// TIA Portal project "read_old_project" (V15.1)

(* hardware
DEVICE "S7-1200 station_1"  S7-1200 Station
   slot 0: "Rack_0"  S7-1200 Rack  Rack  V1.0
   slot 1: "PLC_1"  CPU 1212C DC/DC/DC  6ES7 212-1AE40-0XB0  V4.2
      slot 3: "CB 1241 (RS485)"  CB 1241 (RS485)  6ES7 241-1CH30-1XB0  V1.0
*)

// ===== PLC "PLC_1"  CPU 1212C DC/DC/DC =====

VAR_GLOBAL   // PLC tag table "Default tag table"
   "I0" AT %I0.0 : Bool;
   "I1" AT %I0.1 : Bool;
   "I2" AT %I0.2 : Bool;
   "I3" AT %I0.3 : Bool;
   "distance_raw_1" AT %IW68 : Int;
   "distance_raw_2" AT %IW71 : Int;
   "Conv_power" AT %Q0.0 : Bool;
   "Conv_run" AT %Q0.1 : Bool;
   "Trigger_1" AT %M0.0 : Bool;
   "ChangeApp_1" AT %M0.1 : Bool;
   "AppNo_1" AT %MW2 : UInt;
   "Busy_1" AT %M1.0 : Bool;
   "Done_1" AT %M1.1 : Bool;
   "Error_1" AT %M1.2 : Bool;
   "Status_1" AT %MW4 : Word;
   "ExtStatus_1" AT %MW6 : Word;
   "ActAppNo_1" AT %MW8 : UInt;
   "RcvdLen_1" AT %MW10 : UInt;
   "Connect_1" AT %M0.7 : Bool;
   "Trigger_2" AT %M20.0 : Bool;
   "ChangeApp_2" AT %M20.1 : Bool;
   "Connect_2" AT %M20.7 : Bool;
   "Busy_2" AT %M21.0 : Bool;
   "Done_2" AT %M21.1 : Bool;
   "Error_2" AT %M21.2 : Bool;
   "AppNo_2" AT %MW22 : UInt;
   "Status_2" AT %MW24 : Word;
   "ExtStatus_2" AT %MW26 : Word;
   "ActAppNo_2" AT %MW28 : UInt;
   "RcvdLen_2" AT %MW30 : UInt;
   "System_Byte" AT %MB40 : Byte;
   "FirstScan" AT %M40.0 : Bool;
   "DiagStatusUpdate" AT %M40.1 : Bool;
   "AlwaysTRUE" AT %M40.2 : Bool;
   "AlwaysFALSE" AT %M40.3 : Bool;
   "Clock_Byte" AT %MB41 : Byte;
   "Clock_10Hz" AT %M41.0 : Bool;
   "Clock_5Hz" AT %M41.1 : Bool;
   "Clock_2.5Hz" AT %M41.2 : Bool;
   "Clock_2Hz" AT %M41.3 : Bool;
   "Clock_1.25Hz" AT %M41.4 : Bool;
   "Clock_1Hz" AT %M41.5 : Bool;
   "Clock_0.625Hz" AT %M41.6 : Bool;
   "Clock_0.5Hz" AT %M41.7 : Bool;
   "Edge_1" AT %M1000.0 : Bool;
   "Trigg" AT %M1000.1 : Bool;
   "clear" AT %M1000.2 : Bool;
   "distance_physic_1" AT %MW50 : Int;
   "distance_physic_2" AT %MW52 : Int;
   "M3.3" AT %M3.3 : Bool;
   "Tag_1" AT %M3.4 : Bool;
END_VAR

TYPE "Modbus_Register"
VERSION : 0.1
   STRUCT
      Camera_done : Int;
      Sensor_done : Int;
      Angle : DInt;
      Symetric : Int;
      Conveyor : Int;
      Reset : Int;
      Model : Int;
   END_STRUCT;
END_TYPE

DATA_BLOCK "O2D_Sensor_1"   // DB1
{ S7_Optimized_Access := 'TRUE' }
AUTHOR : ifm-sytl
FAMILY : O2Dxxx
NAME : O2Dxxx_TCP
VERSION : 3.1
// stored: InstanceOfName O2Dxxx_TCP
"O2Dxxx_TCP"
BEGIN
END_DATA_BLOCK

DATA_BLOCK "O2D_Sensor_2"   // DB2
{ S7_Optimized_Access := 'TRUE' }
AUTHOR : ifm-sytl
FAMILY : O2Dxxx
NAME : O2Dxxx_TCP
VERSION : 3.1
// stored: InstanceOfName O2Dxxx_TCP
"O2Dxxx_TCP"
BEGIN
END_DATA_BLOCK

DATA_BLOCK "O2D_Data"   // DB3
{ S7_Optimized_Access := 'TRUE' }
VERSION : 0.1
   VAR
      Response_Sensor_1 : Array[0..127] of Char;
      Response_Sensor_2 : Array[0..63] of Byte;
   END_VAR
BEGIN
END_DATA_BLOCK

DATA_BLOCK "DB_camera"   // DB4
{ S7_Optimized_Access := 'TRUE' }
VERSION : 0.1
   VAR
      Char_reponse : Array[0..127] of Char;
      data_save : Array[0..9] of DInt;
      model_save : Array[0..9] of Int;
      data_convert : DInt;
      data_convert_symetric : DInt;
      count : DInt;
      symetric : Int;
   END_VAR
BEGIN
END_DATA_BLOCK

DATA_BLOCK "DB_modbus"   // DB7
{ S7_Optimized_Access := 'FALSE' }
VERSION : 0.1
   VAR
      Register : "Modbus_Register";
      load_done : Bool;
      load_error : Bool;
      load_status : Word;
      slave_ndr : Bool;
      slave_dr : Bool;
      slave_error : Bool;
      slave_status : Word;
   END_VAR
BEGIN
   Register.Symetric := 1;
END_DATA_BLOCK

FUNCTION_BLOCK "O2Dxxx_TCP"   // FB1, SCL
{ S7_Optimized_Access := 'TRUE' }
AUTHOR : ifm-sytl
FAMILY : O2Dxxx
NAME : O2Dxxx_TCP
VERSION : 3.1
   VAR_INPUT
      LocIF_ID : UInt := 64;
      LocPortNo : UInt := 2000;
      RemIPAddr1 : USInt := 192;
      RemIPAddr2 : USInt := 168;
      RemIPAddr3 : USInt := 0;
      RemIPAddr4 : USInt := 49;
      RemPortNo : UInt := 50010;
      Connect : Bool;
      ConnID : UInt;
      TimeoutTime : Time := T#6S;
      Trigger : Bool;
      ChangeApp : Bool;
      AppNo : UInt := 1;
   END_VAR
   VAR_OUTPUT
      Busy : Bool := TRUE;
      Done : Bool;
      Error : Bool;
      Status : Word;
      ExtStatus : Word;
      ActAppNo : UInt;
      RcvdLen : UInt;
   END_VAR
   VAR_IN_OUT
      Data : Variant;
   END_VAR
   VAR
      fbSend : TSEND;
      fbReceive : TRCV_C;
      tonTimeoutCmd : TON_TIME;
      tonTimeoutPing : TON_TIME;
      tonDlyPing : TON_TIME;
      stConnSet : TCON_IP_v4;
      archRcvBuf : Array[0..33] of Char;
      archSendBuf : Array[0..39] of Char;
      iTicketID : Int;
      iTriggerRespLength : UInt;
      iActAppNo : UInt;
      iRdLength : UInt := 28;
      iRcvFunction : UInt;
      iLeftRcvLength : UInt;
      iBufSize : UInt;
      wStatus : Word;
      wErrorCode : Word;
      wExtErrorCode : Word;
      wErrorCodeConnect : Word;
      wErrorCodeSensor : Word;
      chUserCmdId : Char := '0';
      chCmdId : Char := '0';
      chRcvId : Char;
      xConnEstablished : Bool;
      xReqDisconnect : Bool;
      xReqReconnect : Bool;
      xSendPing : Bool;
      xInitExtRcvBuf : Bool;
      xUserAction : Bool;
      xSensorBlocked : Bool;
      xprevConnect : Bool;
      xprevTrigger : Bool;
      xprevChangeApp : Bool;
      xWaitResponse : Bool;
      xWaitPingResponse : Bool;
      xNewString : Bool;
      xWrToExtBuf : Bool;
      xRcvSysMssgToExt : Bool;
      xBusy : Bool;
      xError : Bool;
      xErrConnect : Bool;
      xErrTimeoutPing : Bool;
      xOutBusy : Bool := TRUE;
      xOutDone : Bool;
      xOutError : Bool;
   END_VAR
   VAR_TEMP
      DISizeOfExtRcvBuf : UDInt;
      DITemp : DInt;
      IDigitFactor : UInt;
      ITemp : Int;
      ICnt : UInt;
      WTemp : Word;
      CHInitValue : Char;
      BInitValue : Byte;
      BCmdId : Byte;
      ARBTemp : Array[0..2] of Byte;
      XRcvBufIsByte : Bool;
      XErrRcvBuf : Bool;
      XNdr : Bool;
      XSysMssgRcvd : Bool;
      XRcvdTicketMatch : Bool;
      XInitDataExch : Bool;
      XreTrigger : Bool;
      XreChangeApp : Bool;
      XErrASCII : Bool;
      XKeepOutput : Bool;
   END_VAR
BEGIN
   // Basic Application program for O2Dx
   // connected to S7 station via CPU-internal Ethernet interface
   // for S7-12xx CPU Firmware V4.1 or higher
   // for S7-15xx CPU Firmware V1.7 or higher

   // Function Block Version 3.1.00

   // With this FB you can
   // - establish TCP/IP V4 connection to the sensor
   // - trigger the sensor and read the result
   // - select active sensor application

   // ---- Inputs ----
   // LocIF_ID      : interface-ID of CPU Ethernet interface (refer to device configuration)
   // LocPortNo     : port.No. in CPU to use for this connection to the sensor (recommended 2000 ff.)
   // RemIPAddr1..4 : IP address of the sensor
   // RemPortNo     : port-No. of sensor process interface
   // Connect       : establish TCP connection to the sensor
   // ConnID        : unique ID as system reference for the connection to the sensor
   // TimeOutTime   : max. waiting time for response from the sensor
   // Trigger       : on rising edge send trigger command to sensor
   // ChangeApp, AppNo : on rising edge of ChangeApp
   //                    activate in AppNo assigned application-No. (3 digits) in the sensor

   // ---- Outputs ----
   // Busy          : no command accepted
   // Done          : command successful completed
   // Error         : error occurred
   // Status        : status information
   // ExtStatus     : extended status information
   // ActAppNo      : active sensor application-No.
   // RcvdLen       : data length in receive buffer

   // ---- In/Outputs ---
   // Data          : pointer to area where to store the data from the sensor


   // ******************************************************************************************************
   // Disclaimer of Warranties

   // ifm disclaims to the fullest extent authorized by law any and all warranties,
   // whether express or implied, including, without limitation,
   // any implied warranties of title, non-infringement, quiet enjoyment,
   // integration, merchantability or fitness for a particular purpose.

   // Without limitation of the foregoing, ifm expressly does not warrant that:
   // (a)  the software will meet your requirements or expectations;
   // (b)  the software or the software content will be free of bugs, errors,
   //      viruses or other defects;
   // (c)  any results, output, or data provided through or generated by the software
   //      will be accurate, up-to-date, complete or reliable;
   // (d)  the software will be compatible with third party software;
   // (e)  any errors in the software will be corrected


   // DEMO SOFTWARE AND TEMPLATES

   // Demo software and templates are provided “as is” and “as available”,
   // without any warranty of any kind, either express or implied.
   // The User acknowledges and agrees to use the software at User’s own risk.
   // In no event shall ifm be held liable for any direct, indirect, incidental
   // or consequential damages arising out of the use of or inability to use the software.
   // User may use the software solely for demonstration purposes
   // and to assess the software functionalities and capabilities.


   // Software written specifically for Customer

   // 1. The software created and used is put together by ifm specially to the customer
   //    using modular software components made by ifm for numerous applications (Standard software modules)
   //    and adapted to the contractual service required (customer-specific application program).

   // 2. Upon complete payment of the purchase price for the customer-specific application program,
   //    ifm transfers the non-exclusive, locally and temporarily unrestricted usage right
   //    thereof to the customer, without the customer acquiring any rights of any kind
   //    to the standard software module on which the individual or customer-specific adaptation is based.
   //    Notwithstanding these provisions, ifm reserves the right to produce and offer
   //    customer specific software solutions of the same kind for other customers
   //    based on other terms of reference. In any case ifm retains a simple right of usage
   //    of the customer–specific solution for internal purposes.

   // 3. Upon acceptance of the program, User acknowledges and agrees to use the software
   //    at User’s own risk. User also acknowledges and agrees upon acceptance of the program
   //    that the software meets the requirements of the specifications agreed upon.
   //    ifm disclaims any and all warranties, in particular regarding fitness of the software
   //    for a particular purpose.
   // ******************************************************************************************************


   // reset error signal
   #xError := #xError AND #xUserAction;  // initialize error signal if no user action active

   // read user inputs
   #XreTrigger := #Trigger AND NOT #xprevTrigger;  // rising edge of input TRIGGER
   #xprevTrigger := #Trigger;  // store state for edge detection
   #XreChangeApp := #ChangeApp AND NOT #xprevChangeApp;  // rising edge of input CHANGE APPLICATION
   #xprevChangeApp := #ChangeApp;  // store state for edge detection
   #xUserAction := (#XreTrigger OR #XreChangeApp) OR #xUserAction;  // set user action started

   // check if user inputs valid
   IF NOT #xError THEN  // no error occurred yet
     IF (#XreTrigger OR #XreChangeApp) AND #xOutBusy THEN
       // command input activated while output BUSY still active
       #xError := TRUE;
       #wErrorCode := 16#8301;  // set error code
       #wExtErrorCode := 0;
     ELSIF (#XreTrigger OR #XreChangeApp) AND NOT #Connect THEN
       // command input activated while input CONNECT = FALSE
       #xError := TRUE;
       #wErrorCode := 16#8302;  // set error code
       #wExtErrorCode := 0;
     ELSIF #XreTrigger AND #XreChangeApp THEN
       // command inputs activated simultaneously
       #xError := TRUE;
       #wErrorCode := 16#8303;  // set error code
       #wExtErrorCode := 0;
     END_IF;
   END_IF;  // check if user inputs valid

   // check external receive buffer is ARRAY OF CHAR or ARRAY OF BYTE
   #DISizeOfExtRcvBuf := CountOfElements(#Data);  // get size of external receive buffer
   #XErrRcvBuf := #DISizeOfExtRcvBuf = 0;  // check if external receive buffer is an array
   IF NOT #XErrRcvBuf THEN
     // external is an array
     #XRcvBufIsByte := TypeOfElements(#Data) = Byte;  // check if element data type of external receive buffer is BYTE
     #XErrRcvBuf := TypeOfElements(#Data) <> Char AND NOT #XRcvBufIsByte;  // check element data type of receive buffer is valid
   END_IF;
   IF #XErrRcvBuf AND NOT #xError THEN
     // external receive buffer invalid (only ARRAY of BYTE or ARRAY of CHAR are valid)
     #xError := TRUE;
     #wErrorCode := 16#8101;  // set error code
     #wExtErrorCode := 0;
   END_IF;

   // initialize external receive buffer
   #xInitExtRcvBuf := #XreTrigger OR #XreChangeApp OR #xInitExtRcvBuf;  // initialize external receive buffer
   IF #xInitExtRcvBuf AND NOT #XErrRcvBuf THEN
     #CHInitValue := ' ';  // set initial value for external receive buffer
     #BInitValue := 0;
     FOR #DITemp := 0 TO UDINT_TO_DINT(#DISizeOfExtRcvBuf) - 1 DO  // loop complete external receive buffer
       IF #XRcvBufIsByte THEN  // initialize external receive buffer with initial BYTE value
         #ITemp := MOVE_BLK_VARIANT(SRC := #BInitValue, SRC_INDEX := 0, DEST => #Data, DEST_INDEX := #DITemp, COUNT := 1);
       ELSE  // initialize external receive buffer with initial CHAR value
         #ITemp := MOVE_BLK_VARIANT(SRC := #CHInitValue, SRC_INDEX := 0, DEST => #Data, DEST_INDEX := #DITemp, COUNT := 1);
       END_IF;
       IF #ITemp <> 0 THEN  // error by access to external receive buffer
         IF NOT #xError THEN
           #xError := TRUE;
           #wErrorCode := 16#8400;  // set error code
           #wExtErrorCode := INT_TO_WORD(#ITemp);
         END_IF;
         EXIT;  // abort initialisation
       END_IF;
     END_FOR;
     #xInitExtRcvBuf := FALSE;  // reset request
   END_IF;  // initialize external receive buffer

   // set connection parameter
   IF #Connect AND NOT #xprevConnect THEN  // rising edge of input CONNECT
     // fill TCP/IP V4 connection structure
     #stConnSet.InterfaceId := #LocIF_ID;  // set hardware identifier of local interface (see CPU device properties )
     #stConnSet.ID := UINT_TO_WORD(#ConnID);  // set reference to this connection
     #stConnSet.ConnectionType := 17;  // set connection type = TCP
     #stConnSet.ActiveEstablished := TRUE;  // set active connection establishment
     #stConnSet.RemoteAddress.ADDR[1] := USINT_TO_BYTE(#RemIPAddr1);  // set IP address of remote connection partner
     #stConnSet.RemoteAddress.ADDR[2] := USINT_TO_BYTE(#RemIPAddr2);
     #stConnSet.RemoteAddress.ADDR[3] := USINT_TO_BYTE(#RemIPAddr3);
     #stConnSet.RemoteAddress.ADDR[4] := USINT_TO_BYTE(#RemIPAddr4);
     #stConnSet.RemotePort := #RemPortNo;  // set port address of remote connection partner
     #stConnSet.LocalPort := #LocPortNo;  // set local port address
   END_IF;  // rising edge of input CONNECT
   #xprevConnect := #Connect;  // store state for edge detection

   #xReqDisconnect := NOT #Connect AND #xConnEstablished OR #xReqDisconnect;  // set request to disconnect
   #xConnEstablished := #xConnEstablished AND NOT #xReqDisconnect AND NOT #xReqReconnect;  // reset connection established

   #fbReceive.CONT := #Connect AND NOT #xReqDisconnect AND NOT #xReqReconnect;  // establish connection
   #fbReceive.EN_R := TRUE;  // enable receive data
   #fbReceive.ADHOC := FALSE;  // disable AdHoc-mode
   #fbReceive.LEN := #iRdLength;  // set length to receive

   // receive data
   IF #xWrToExtBuf THEN  // select receive buffer
     // write to external receive buffer
     #fbReceive(CONNECT := #stConnSet,
                DATA := #Data);
   ELSE  // select receive buffer
     // write to internal receive buffer
     #fbReceive(CONNECT := #stConnSet,
                DATA := #archRcvBuf);
   END_IF;  // select receive buffer

   // result disconnect
   IF #fbReceive.STATUS = 16#7000 OR #fbReceive.STATUS = 16#0003 OR // disconnecting done
     #fbReceive.STATUS = 16#80A3  // no connection established
   THEN
     // disconnected successfully
     #xReqDisconnect := FALSE;  // reset request to disconnect
     #xReqReconnect := FALSE;  // reset request to reconnect
   END_IF;  // result disconnect

   // result connect
   IF NOT #Connect THEN  // reset error connect
     // reset error establish connection and timeout
     #xErrConnect := FALSE;
     #xErrTimeoutPing := FALSE;
     #xSensorBlocked := FALSE;
   ELSIF #fbReceive.CONT AND NOT #xConnEstablished AND #fbReceive.ERROR AND #fbReceive.STATUS <> 16#80C4 THEN
     // set error establish connection      
     #xErrConnect := TRUE;
     #xReqDisconnect := TRUE;
     #wErrorCodeConnect := #fbReceive.STATUS;  // save error code
   ELSIF #fbReceive.CONT AND NOT #xConnEstablished AND
     (#fbReceive.STATUS = 16#7004 OR #fbReceive.STATUS = 16#7006 OR #fbReceive.STATUS = 16#0001) THEN
     // connection established successfully
     #xConnEstablished := TRUE;
     #xErrConnect := FALSE;
     #xErrTimeoutPing := FALSE;
     #chCmdId := '1';  // execute command "v03"
   END_IF;  // result establish connection
   IF #xErrConnect AND NOT #xErrTimeoutPing AND NOT #xError THEN
     // set error code for error by establishing connection
     #xError := TRUE;
     #wErrorCode := 16#8201;  // set error code
     #wExtErrorCode := #wErrorCodeConnect;  // show error code of FB
   END_IF;  // error code establish connection

   // result receive data
   #XNdr := NOT #fbReceive.BUSY AND #fbReceive.DONE;  // new data received
   IF #fbReceive.CONT AND NOT #fbReceive.BUSY AND #fbReceive.ERROR THEN
     // error receive data
     #xReqReconnect := TRUE;  // set request disconnect
     IF NOT #xError AND #xBusy THEN
       #xError := TRUE;  // set error occurred
       #wErrorCode := 16#8203;  // set error code
       #wExtErrorCode := #fbReceive.STATUS;  // show error code of receive block
     END_IF;  // set error code
   END_IF;  // error receive data

   // cancel waiting for response
   IF NOT #fbReceive.CONT THEN
     #xWaitResponse := FALSE;
     #xWaitPingResponse := FALSE;
   END_IF;

   // timeout
   #tonTimeoutCmd(IN := #xWaitResponse AND #fbReceive.BUSY AND #xConnEstablished,
                  PT := #TimeoutTime);
   IF #tonTimeoutCmd.Q THEN
     // no response from sensor within surveillance time
     // (also happen if response string is shorter than expected;
     // the receive block will not provide data as long the buffer is not full yet)
     #xReqReconnect := TRUE;  // set request reconnect
     IF NOT #xError THEN
       #xError := TRUE;  // set error occurred
       #wErrorCode := 16#8205;  // set error code
       #wExtErrorCode := 0;
     END_IF;  // set error code
   END_IF;  // error receive data

   #XInitDataExch := NOT #xConnEstablished;  // preset request initialize data exchange

   IF #XNdr AND NOT #XInitDataExch THEN  // new data received

     #iLeftRcvLength := #iLeftRcvLength - UDINT_TO_UINT(#fbReceive.RCVD_LEN);  // update remaining length to receive

     CASE #iRcvFunction OF  // receive function selector

       0:  //receive 28 byte until "<CR><LF>10" received
         // look for "<CR><LF>10" in received data;
         // if found activate receive byte-wise

         FOR #ITemp := 0 TO 24 DO  // 25 possible DWORDs to check
           IF #archRcvBuf[#ITemp] = '$R' AND #archRcvBuf[#ITemp + 1] = '$L' AND
             #archRcvBuf[#ITemp + 2] = '1' AND #archRcvBuf[#ITemp + 3] = '0' THEN  // "<CR><LF>10" found

             // prepare FOR receiving the rest Byte-wise
             #xWaitResponse := FALSE;
             #iRdLength := 1;  // set length to receive
             #iRcvFunction := 1;  // activate receive function 1
           END_IF;  // "<CR><LF>10" found
         END_FOR;  // 25 possible DWORDs to check

       1:  // receive byte-wise until protocol V03 approved
         // check for response = ..."1003*<CR><LF>" to confirm protocol V03 is active

         #archRcvBuf[28] := #archRcvBuf[0];  // copy received byte to end of received data

         // shift received data in buffer 1 byte to left
         FOR #ITemp := 0 TO 27 DO
           #archRcvBuf[#ITemp] := #archRcvBuf[#ITemp + 1];
         END_FOR;

         // check for "1003" and "<CR><LF>"
         IF #archRcvBuf[21] = '1' AND #archRcvBuf[22] = '0' AND #archRcvBuf[23] = '0' AND #archRcvBuf[24] = '3' AND
           #archRcvBuf[26] = '$R' AND #archRcvBuf[27] = '$L' THEN  // "1003" and "<CR><LF>" received

           // response to command "v03" received
           IF #archRcvBuf[25] <> '*' THEN  // check acknowledge
             // protocol V03 not acknowledged
             IF NOT #xError THEN  // error protocol V03
               #xError := TRUE;
               #wErrorCode := 16#8001;  // set error code
               #wExtErrorCode := 0;
             END_IF;  // error protocol V03
             #XInitDataExch := TRUE;
           ELSE  // check acknowledge
             // protocol V03 acknowledged
             #chCmdId := '8';  // execute command "a?"
             #iLeftRcvLength := 0;  // no more data to receive
             #iRcvFunction := 4;  // complete command
           END_IF;  // check acknowledge

         END_IF;  // "1003" and "<CR><LF>" received

       2:  // evaluate ID and length information
         // identify length information and response-ID;
         // check if payload is to receive with or without evaluation

         #XErrASCII := #archRcvBuf[4] <> 'L' OR
         #archRcvBuf[5] <> '0' OR #archRcvBuf[6] <> '0' OR #archRcvBuf[7] <> '0' OR #archRcvBuf[8] <> '0' OR
         #archRcvBuf[15] <> '$L';  // check begin and end of length information string

         // convert length from ASCII to UINT
         #IDigitFactor := 10000;  // set digit factor
         #iLeftRcvLength := 0;  // initialize remaining length to receive
         FOR #ITemp := 9 TO 13 DO  // loop lowest 5 length information digits
           IF #archRcvBuf[#ITemp] < '0' OR #archRcvBuf[#ITemp] > '9' THEN  // check for ASCII range 0..9
             // out of range
             #XErrASCII := TRUE;  // set error ASCII data
           ELSE  // check for ASCII range 0..9
             // calculate response length
             #iLeftRcvLength := (CHAR_TO_UINT(#archRcvBuf[#ITemp]) - 48) * #IDigitFactor + #iLeftRcvLength;
           END_IF;  // check for ASCII range 0..9
           #IDigitFactor := #IDigitFactor / 10;  // update digit factor for next digit
         END_FOR; // loop lowest 5 length information digits

         IF #XErrASCII THEN  // error in length information data
           // error in ASCII data of length information string
           IF NOT #xError THEN  // no error yet
             #xError := TRUE;
             #wErrorCode := 16#8402;  // set error code
             #wExtErrorCode := 0;
           END_IF;  // no error yet
           // synchronize data exchange
           #XInitDataExch := TRUE;  // enable initialize data exchange
           #chCmdId := '1';  // execute command "v03"
         ELSE  // error in length information data
           // length information extracted successfully
           // prepare to receive payload data

           // correct left length to receive
           #iLeftRcvLength := #iLeftRcvLength - 4;  // 4 Byte ticket-No. is received already

           // evaluate received command-ID and ticket-No.
           #chRcvId := #archRcvBuf[0];  // store received command-ID
           #XSysMssgRcvd := #archRcvBuf[0] = '0' AND #archRcvBuf[1] = '0' AND #archRcvBuf[2] = '0' AND #archRcvBuf[3] = '0';  // check response-ID
           #XRcvdTicketMatch := #archRcvBuf[0] = #archSendBuf[0] AND
           #archRcvBuf[1] = #archSendBuf[1] AND
           #archRcvBuf[2] = #archSendBuf[2] AND
           #archRcvBuf[3] = #archSendBuf[3];  // received ticket-No. match to last sent ticket-No.
           #xWaitResponse := #xWaitResponse AND NOT #XRcvdTicketMatch;  // reset wait for response if response of command is received

           // select receive buffer for payload data to receive
           #xRcvSysMssgToExt := #XSysMssgRcvd AND NOT #xSensorBlocked AND NOT #Trigger AND NOT #ChangeApp AND NOT #xError;
           #xInitExtRcvBuf := (#xRcvSysMssgToExt OR #XRcvdTicketMatch AND #chRcvId = '9') AND NOT #XErrRcvBuf;
           #xWrToExtBuf := #xInitExtRcvBuf AND #iLeftRcvLength <> 3;
           IF #xWrToExtBuf THEN  // select receive buffer
             // use external receive buffer
             #iBufSize := UDINT_TO_UINT(#DISizeOfExtRcvBuf);  // set receive buffer size to size of external buffer
             #iTriggerRespLength := #iLeftRcvLength;  // store received payload data length
           ELSE  // select receive buffer
             // use internal receive buffer
             #iBufSize := 34;  // set receive buffer size to size of internal buffer
             #iTriggerRespLength := 0;  // initialize received payload data length
           END_IF;  // select receive buffer

           #iRdLength := MIN(IN1 := #iLeftRcvLength, IN2 := #iBufSize);  // limit receive length to receive buffer size
           #xNewString := TRUE;  // set new string will be received

           // select next receive function
           IF NOT #XRcvdTicketMatch AND NOT #xSensorBlocked OR #xWrToExtBuf THEN
             #iRcvFunction := 4;  // receive data without evaluation
           ELSE
             #iRcvFunction := 3;  // receive data to evaluate
           END_IF;  // select next receive function

         END_IF;  // error in length information data

       3:  // evaluate response data
         IF #chRcvId = '0' THEN
           // ping response received
           IF NOT #xUserAction AND #archRcvBuf[0] = '!' THEN
             // sensor used by another application (GUI)
             #xSensorBlocked := TRUE;
           ELSIF NOT #xUserAction THEN
             // sensor available
             IF #xSensorBlocked THEN  // sensor was unavailable
               #chCmdId := '8';  // execute command "a?"
               #xSensorBlocked := FALSE;
             END_IF;  // sensor available
           END_IF;  // ping response received

         ELSIF #fbReceive.RCVD_LEN = 3 AND #archRcvBuf[0] = '?' AND #archRcvBuf[1] = '$R' AND #archRcvBuf[2] = '$L' THEN
           // sensor returns "command unknown"
           IF NOT #xError THEN
             // error command unknown
             #xError := TRUE;
             #wErrorCode := 16#8300;  // set error code
             #wExtErrorCode := 0;
           END_IF;  // error command unknown

         ELSIF #fbReceive.RCVD_LEN = 3 AND #archRcvBuf[0] = '!' AND #archRcvBuf[1] = '$R' AND #archRcvBuf[2] = '$L' THEN
           // sensor returns "unable to execute command"
           // get error code from sensor
           #chCmdId := '2';  // execute command "E?"
         ELSE
           // data to evaluate received
           // evaluate received data of each command special
           CASE CHAR_TO_INT(#chRcvId) - 48 OF  // convert ASCII to integer

             2:  // evaluate response to command "E?"
               // error code from sensor received
               #wErrorCodeSensor.%B1 := INT_TO_BYTE((CHAR_TO_INT(#archRcvBuf[0]) - 48) * 16 + (CHAR_TO_INT(#archRcvBuf[1]) - 48));  // convert hi-byte of error code
               #wErrorCodeSensor.%B0 := INT_TO_BYTE((CHAR_TO_INT(#archRcvBuf[2]) - 48) * 16 + (CHAR_TO_INT(#archRcvBuf[3]) - 48));  // convert low-byte of error code
               IF #xUserAction AND NOT #xError THEN
                 // error sensor unable to execute command
                 #xError := TRUE;
                 #wErrorCode := 16#8000;  // set error code
                 #wExtErrorCode := #wErrorCodeSensor;  // show error code from sensor
               END_IF;  // error sensor unable to execute command
               #chCmdId := '8';  // execute command "a?"

             4:  // evaluate response to command "c + group and application-No."
               #chCmdId := '8';  // execute command "a?"

             8:  // evaluate response to command "a?"
               // extract number of active configuration and convert ASCII to integer
               #iActAppNo := (CHAR_TO_UINT(#archRcvBuf[5]) - 48) * 10 + CHAR_TO_UINT(#archRcvBuf[6]) - 48;

             9:  // evaluate response to command "T?"
               // response length = 3 characters but not a negative acknowledge;
               // then copy received data into external receive buffer
               IF #XRcvBufIsByte THEN  // element data type of external receive buffer is BYTE
                 // convert data type and copy to external receive buffer
                 #ARBTemp[0] := CHAR_TO_BYTE(#archRcvBuf[0]);
                 #ARBTemp[1] := CHAR_TO_BYTE(#archRcvBuf[1]);
                 #ARBTemp[2] := CHAR_TO_BYTE(#archRcvBuf[2]);
                 #ITemp := MOVE_BLK_VARIANT(SRC := #ARBTemp, SRC_INDEX := 0, DEST => #Data, DEST_INDEX := 0, COUNT := 3);
               ELSE  // copy to external receive buffer
                 #ITemp := MOVE_BLK_VARIANT(SRC := #archRcvBuf, SRC_INDEX := 0, DEST => #Data, DEST_INDEX := 0, COUNT := 3);
               END_IF;
               IF #ITemp = 0 THEN  // copy data successful
                 #iTriggerRespLength := 3;  // store received payload data length
               ELSIF NOT #xError THEN
                 // error by access to external receive buffer
                 #xError := TRUE;
                 #wErrorCode := 16#8400;  // set error code
                 #wExtErrorCode := INT_TO_WORD(#ITemp);
               END_IF;

           END_CASE;  // evaluate received data of each command special
         END_IF;  // evaluate response data
         #iRcvFunction := 4;  // evaluation finished, receive rest of response data

     END_CASE;  // receive function selector

     // receive data without evaluation
     IF #iRcvFunction = 4 AND NOT #XInitDataExch THEN  // receive function 4 active

       // receive data without evaluation
       IF #iLeftRcvLength > 0 THEN  // receiving data completed?
         // not all data received yet
         IF NOT #xNewString AND #xWrToExtBuf THEN
           // external buffer full
           IF NOT #xError THEN  // error external receive buffer too small
             #xError := TRUE;
             #wErrorCode := 16#8401;  // set error code
             #wExtErrorCode := UINT_TO_WORD(#iTriggerRespLength);  // show trigger response length
           END_IF;  // error external receive buffer too small
           #xWrToExtBuf := FALSE;  // change to internal receive buffer
           #iBufSize := 34;  // set size of used buffer
         END_IF;  // external buffer full
         #iRdLength := MIN(IN1 := #iLeftRcvLength, IN2 := #iBufSize);  // limit receive length
         #xNewString := FALSE;  // reset new string to receive

       ELSE  // receiving data completed?
         // all data received
         #xWrToExtBuf := FALSE;  // activate internal receive buffer
         #xBusy := #xBusy AND (#xWaitResponse OR #chRcvId = '0');  // enable new command, except Ping response is received
         #iRdLength := 20;  // set length 16 byte length information string + 4 byte ticket-No.
         #iRcvFunction := 2;  // activate receive function 2
       END_IF;  // receiving data completed?
     END_IF;  // receive function 4 active

   END_IF;  // new data received

   // initialize data exchange
   IF #XInitDataExch THEN
     // prepare for receiving response to command "v03"
     #xBusy := FALSE;
     #xWrToExtBuf := FALSE;
     #xRcvSysMssgToExt := FALSE;
     #iRdLength := 28; // set initial length to read
     #iRcvFunction := 0;  // activate receive function 0
   END_IF;  // initialize data exchange

   //**************************************************************
   // after certain time of inactivity send ping command to check connection
   #tonDlyPing(IN := (#iRcvFunction = 2 OR #xSensorBlocked) AND #fbReceive.BUSY AND NOT #xBusy AND NOT #xSendPing,
               PT := t#3s,  // inactivity time
               Q => #xSendPing);  // activate send ping command

   // timeout ping
   #xWaitPingResponse := #xWaitPingResponse AND NOT #XNdr AND #xConnEstablished;  // any received data reset ping timeout
   #tonTimeoutPing(IN := #xWaitPingResponse,
                   PT := t#1s);
   IF #tonTimeoutPing.Q THEN
     #xErrTimeoutPing := TRUE;  // timeout ping occurred
     #xReqReconnect := TRUE;  // set request reconnect
   END_IF;
   IF #xErrTimeoutPing AND NOT #xError THEN  // error timeout ping
     #xError := TRUE;  // set error occurred
     #wErrorCode := 16#8206;  // set error code
     #wExtErrorCode := 0;
   END_IF;  // error timeout ping

   //**************************************************************
   // request send command
   IF #XreTrigger THEN
     #chUserCmdId := '9';  // store user requested command-ID
   END_IF;
   IF #XreChangeApp THEN
     #chUserCmdId := '4';  // store user requested command-ID
   END_IF;
   IF (#XreTrigger OR #XreChangeApp) AND NOT #xError THEN
     #chCmdId := #chUserCmdId;  // apply requested command
   END_IF;
   #xBusy := #chCmdId <> '0' OR #xBusy;  // if command requested then set busy

   #fbSend.REQ := (#chCmdId <> '0' OR #xSendPing) AND #xConnEstablished AND NOT #fbSend.BUSY;  // activate sending data
   IF #fbSend.REQ THEN  // build command to send

     // create new ticket-ID
     IF #iTicketID > 0 AND #iTicketID < 999 THEN
       #iTicketID := #iTicketID + 1;  // increase ticket-ID
     ELSE  // limit reached
       #iTicketID := 1;  // initialize ticket-ID
     END_IF;

     // fill most common parts into send buffer
     #archSendBuf[0] := #chCmdId;  // command-ID
     #archSendBuf[1] := INT_TO_CHAR(#iTicketID / 100 + 48);  // convert 100th digit of ticket-ID to ASCII
     #ITemp := #iTicketID - #iTicketID / 100 * 100;  // get rest of division
     #archSendBuf[2] := INT_TO_CHAR(#ITemp / 10 + 48);  // convert 10th digit of ticket-ID to ASCII
     #ITemp := #ITemp - #ITemp / 10 * 10;  // get rest of division
     #archSendBuf[3] := INT_TO_CHAR(#ITemp + 48);  // convert 1th digit of ticket-ID to ASCII
     #archSendBuf[4] := 'L';
     FOR #ITemp := 5 TO 12 DO  // preset length information with "0"
       #archSendBuf[#ITemp] := '0';
     END_FOR;
     #archSendBuf[13] := '8';  // preset most common command length = 8 bytes
     #archSendBuf[14] := '$R';  // "<CR>"
     #archSendBuf[15] := '$L';  // "<LF>"
     #archSendBuf[16] := #archSendBuf[0];  // repeat ticket-No.
     #archSendBuf[17] := #archSendBuf[1];
     #archSendBuf[18] := #archSendBuf[2];
     #archSendBuf[19] := #archSendBuf[3];
     FOR #ITemp := 20 TO 39 DO  // preset rest of send buffer with " "
       #archSendBuf[#ITemp] := ' ';
     END_FOR;

     // select command
     CASE CHAR_TO_INT(#chCmdId) - 48 OF  // convert ASCII to integer

       0:  // command "s?" as ping command 
         #archSendBuf[20] := 's';
         #archSendBuf[21] := '?';
         #archSendBuf[22] := '$R';  // "<CR>"
         #archSendBuf[23] := '$L';  // "<LF>"
         #fbSend.LEN := 24;  // set length to send

       1:  // command "v03" in all protocol versions
         // "v03<CR><LF>" for protocol 1 and 4
         // "1002v03<CR><LF>" for protocol 2
         // "1003L000000009<CR><LF>1003v03<CR><LF>" for protocol 3
         Strg_TO_Chars(Strg := 'v03$R$L1002v03$R$L1003L000000009$R$L1003v03$R$L',  // source string
                       Chars := #archSendBuf,  // destination array
                       pChars := 0,  // destination start index
                       Cnt => #ICnt);  // number of copied characters
         #fbSend.LEN := UINT_TO_UDINT(#ICnt);  // set length to send

       2:  // command "E?"
         #archSendBuf[20] := 'E';
         #archSendBuf[21] := '?';
         #archSendBuf[22] := '$R';  // "<CR>"
         #archSendBuf[23] := '$L';  // "<LF>"
         #fbSend.LEN := 24;  // set length to send

       4:  // command "c + group-No. + application-No."
         #archSendBuf[12] := '1';  // overwrite preset payload data length
         #archSendBuf[13] := '0';  // command length = 10 bytes
         #archSendBuf[20] := 'c';
         #archSendBuf[21] := UINT_TO_CHAR(#AppNo / 100 + 48);  // convert 100th digit of input APPLICATION-NO. to ASCII
         #ITemp := UINT_TO_INT(#AppNo - #AppNo / 100 * 100);  // get rest of division
         #archSendBuf[22] := INT_TO_CHAR(#ITemp / 10 + 48);  // convert 10th digit of APPLICATION-NO. to ASCII
         #ITemp := #ITemp - #ITemp / 10 * 10;  // get rest of division
         #archSendBuf[23] := INT_TO_CHAR(#ITemp + 48);  // convert 1th digit of APPLICATION-NO. to ASCII
         #archSendBuf[24] := '$R';  // "<CR>"
         #archSendBuf[25] := '$L';  // "<LF>"
         #fbSend.LEN := 26;  // set length to send

       8:  // command "a?"
         #archSendBuf[20] := 'a';
         #archSendBuf[21] := '?';
         #archSendBuf[22] := '$R';  // "<CR>"
         #archSendBuf[23] := '$L';  // "<LF>"
         #fbSend.LEN := 24;  // set length to send

       9:  // command "T?"
         #archSendBuf[20] := 'T';
         #archSendBuf[21] := '?';
         #archSendBuf[22] := '$R';  // "<CR>"
         #archSendBuf[23] := '$L';  // "<LF>"
         #fbSend.LEN := 24;  // set length to send

       ELSE  // unknown command-ID
         #fbSend.REQ := FALSE;  // reset send request
     END_CASE;  // select command

     // command is build
     #xWaitPingResponse := #fbSend.REQ AND #chCmdId = '0';  // set wait for ping response
     #xWaitResponse := #fbSend.REQ AND NOT #xWaitPingResponse;  // set wait for command response
     #chCmdId := '0';  // initialize command-ID
   END_IF;  // build command to send

   // send data
   #fbSend(ID := #stConnSet.ID,
           DATA := #archSendBuf);  // send data

   // check send result
   IF #fbSend.ERROR AND #archSendBuf[0] <> '0' THEN
     // error while sending data
     #xReqReconnect := TRUE;  // set request reconnect
     IF NOT #xError THEN
       #xError := TRUE;
       #wErrorCode := 16#8204;  // set error code
       #wExtErrorCode := #fbSend.STATUS;  // show error code of send block
     END_IF;  // send error
   END_IF;  // send result

   // build internal status code
   IF NOT #Connect AND (#fbReceive.STATUS = 16#7000 OR #fbReceive.STATUS = 16#0003) THEN
     #wStatus := 16#1000;  // disconnected
   ELSIF #xReqDisconnect OR #xReqReconnect THEN
     #wStatus := 16#1001;  // disconnecting in progress
   ELSIF #Connect AND NOT #xConnEstablished THEN
     #wStatus := 16#1002;  // connecting in progress
   ELSIF #iRcvFunction < 2 THEN
     // synchronisation phase
     IF #fbSend.BUSY THEN
       #wStatus := 16#2001;  // send command "v03"
     ELSIF #iRcvFunction = 0 THEN
       #wStatus := 16#2002;
     ELSE
       #wStatus := 16#2003;
     END_IF;
     // end synchronisation phase
   ELSIF #xSensorBlocked THEN
     #wStatus := 16#3000;  // sensor unavailable
   ELSE
     // data exchange phase
     IF NOT #xBusy AND #iRcvFunction = 2 THEN
       #wStatus := 16#7000;
     ELSIF #fbSend.BUSY THEN
       #wStatus := 16#7001;  // send data active
     ELSE
       #wStatus := 16#7000 OR UINT_TO_WORD(#iRcvFunction);
     END_IF;
     IF #xBusy THEN
       #BCmdId := INT_TO_BYTE(CHAR_TO_INT(#archSendBuf[0]) - 48);  // convert ASCII to byte
       #wStatus.%B1 := #wStatus.%B1 OR #BCmdId;  // add active command-ID
     END_IF;
     // end data exchange phase
   END_IF;  // build internal status code

   // output BUSY
   #xOutBusy := #xBusy OR #iRcvFunction < 2 OR NOT #xConnEstablished OR #xReqReconnect OR #xSensorBlocked;
   #Busy := #xOutBusy;

   // keep output DONE and ERROR as long the triggering input still active
   #XKeepOutput := (#chUserCmdId = '9' AND #Trigger OR #chUserCmdId = '4' AND #ChangeApp) AND NOT #XreTrigger AND NOT #XreChangeApp;

   // output DONE
   #xOutDone := (#iRcvFunction = 2 AND #xRcvSysMssgToExt  // receive system message to ext. buffer finished
   OR #xUserAction  // user action started
   ) AND NOT #xBusy AND NOT #xError AND NOT #XErrRcvBuf // no command in progress and no error
   OR #xOutDone AND #XKeepOutput;  // keep output as long triggering input still set
   #Done := #xOutDone;

   // output ERROR
   #xOutError := (#xError OR #XErrRcvBuf) AND NOT #xBusy AND NOT #xOutDone  // error occurred and no command in progress
   OR #xOutError AND #XKeepOutput;  // keep output as long triggering input still set
   #Error := #xOutError;

   // output STATUS and EXTSTATUS
   IF #xOutDone THEN
     // if output DONE is set, show STATUS = 0x0000, EXTSTATUS = internal status code
     #Status := 16#0000;
     #ExtStatus := #wStatus;
   ELSIF #xOutError THEN
     // if output ERROR is set, show error codes STATUS and EXTSTATUS
     #Status := #wErrorCode;
     #ExtStatus := #wExtErrorCode;
   ELSE
     // else show STATUS = internal status code, EXTSTATUS = status of receive block
     #Status := #wStatus;
     #ExtStatus := #fbReceive.STATUS;
   END_IF;  // end output STATUS

   // output ACTIVE APPLICATION-NO. in the sensor
   IF NOT #xConnEstablished OR #xSensorBlocked THEN
     #iActAppNo := 0;  // reset active application 
   END_IF;
   #ActAppNo := #iActAppNo;

   // output DATA LENGTH in external receive buffer
   IF #XreTrigger OR #XreChangeApp OR #xInitExtRcvBuf OR #XErrRcvBuf THEN
     #RcvdLen := 0;
   ELSIF #xOutDone AND (#xUserAction OR #xRcvSysMssgToExt) THEN
     #RcvdLen := #iTriggerRespLength;
   END_IF;

   #xUserAction := #xUserAction AND #xBusy;  // reset user action started

   // reset receive system message to external receive buffer
   #xRcvSysMssgToExt := #xRcvSysMssgToExt AND NOT #xOutDone;  // reset if output DONE is set
END_FUNCTION_BLOCK

FUNCTION "Angle_Convert_Push" : Void   // FC1, LAD
{ S7_Optimized_Access := 'TRUE' }
VERSION : 0.1
   VAR_TEMP
      Temp_1 : DInt;
      Temp_2 : DInt;
      Temp_3 : DInt;
      Temp_4 : DInt;
      Temp_5 : DInt;
      Temp_6 : DInt;
   END_VAR
BEGIN

REGION Network 1 (SCL)
   //Convert
   #Temp_1 := CHAR_TO_DINT("DB_camera".Char_reponse[33]);
   #Temp_2 := CHAR_TO_DINT("DB_camera".Char_reponse[34]);
   #Temp_3 := CHAR_TO_DINT("DB_camera".Char_reponse[35]);
   #Temp_4 := CHAR_TO_DINT("DB_camera".Char_reponse[36]);
   #Temp_5 := CHAR_TO_DINT("DB_camera".Char_reponse[37]);
   #Temp_6 := CHAR_TO_DINT("DB_camera".Char_reponse[38]);

   "DB_camera".data_convert := (#Temp_2 - 48) * 10000000 + (#Temp_3 - 48) * 1000000 + (#Temp_4 - 48) * 100000 + (#Temp_6 - 48) * 10000;
   IF #Temp_1 = 43 THEN
       "DB_camera".data_convert := "DB_camera".data_convert * (-1);
   END_IF;
   //Push //symetric 1=rectang//2=square
   IF ("DB_camera".data_convert >= -18000000) AND ("DB_camera".data_convert <= 18000000) THEN
       #Temp_1 := CHAR_TO_DINT("DB_camera".Char_reponse[33]);
       IF "DB_modbus".Register.Symetric = 0 THEN
           "DB_camera".data_convert_symetric := "DB_camera".data_convert;
       ELSIF "DB_modbus".Register.Symetric = 1 THEN
           IF "DB_camera".data_convert > 9000000 THEN
               "DB_camera".data_convert_symetric := "DB_camera".data_convert - 18000000;
           ELSIF "DB_camera".data_convert < -9000000 THEN
               "DB_camera".data_convert_symetric := "DB_camera".data_convert + 18000000;
           ELSE
               "DB_camera".data_convert_symetric := "DB_camera".data_convert;
           END_IF;
       ELSIF "DB_modbus".Register.Symetric = 2 THEN
           IF "DB_camera".data_convert > 4500000 AND "DB_camera".data_convert <= 13500000 THEN
               "DB_camera".data_convert_symetric := "DB_camera".data_convert - 9000000;
           ELSIF "DB_camera".data_convert < -4500000 AND "DB_camera".data_convert >= -13500000 THEN
               "DB_camera".data_convert_symetric := "DB_camera".data_convert + 9000000;
           ELSIF "DB_camera".data_convert > 13500000 THEN
               "DB_camera".data_convert_symetric := "DB_camera".data_convert - 18000000;
           ELSIF "DB_camera".data_convert < -13500000 THEN
               "DB_camera".data_convert_symetric := "DB_camera".data_convert + 18000000;
           ELSE
               "DB_camera".data_convert_symetric := "DB_camera".data_convert;
           END_IF; 
       END_IF;

       "DB_camera".count := "DB_camera".count + 1;
       "DB_camera".data_save["DB_camera".count - 1] := "DB_camera".data_convert_symetric;
       "DB_camera".model_save["DB_camera".count - 1] := CHAR_TO_DINT("DB_camera".Char_reponse[21]) - 48;
   END_IF;
END_REGION
END_FUNCTION

FUNCTION "Angle_Mov_Pull" : Void   // FC2, LAD
{ S7_Optimized_Access := 'TRUE' }
VERSION : 0.1
   VAR_TEMP
      forloop : DInt;
   END_VAR
BEGIN

REGION Network 1 (SCL)
   IF ("DB_camera".data_save[0] >= -18000000) AND ("DB_camera".data_save[0] <= 18000000) THEN
       //mov
       "DB_modbus".Register.Angle := "DB_camera".data_save[0];
       "DB_modbus".Register.Model := "DB_camera".model_save[0];
       "DB_modbus".Register.Camera_done := 1;

       //pull
       "DB_camera".count := "DB_camera".count - 1;
       FOR #forloop := 0 TO ("DB_camera".count - 1) DO
           "DB_camera".data_save[#forloop] := "DB_camera".data_save[#forloop + 1];
           "DB_camera".model_save[#forloop] := "DB_camera".model_save[#forloop + 1];
       END_FOR;
       "DB_camera".data_save["DB_camera".count] := -177760000;
       "DB_camera".model_save["DB_camera".count] := 0;
   END_IF;
END_REGION
END_FUNCTION

ORGANIZATION_BLOCK "Main"   // OB1, LAD, ProgramCycle
{ S7_Optimized_Access := 'TRUE' }
VERSION : 0.1
   VAR_INPUT
      Initial_Call : Bool;
      Remanence : Bool;
   END_VAR
   VAR_TEMP   // added for the SCL form of the ladder/FBD networks
      _w1 : Bool;
   END_VAR
BEGIN

REGION Network 1: Camera1
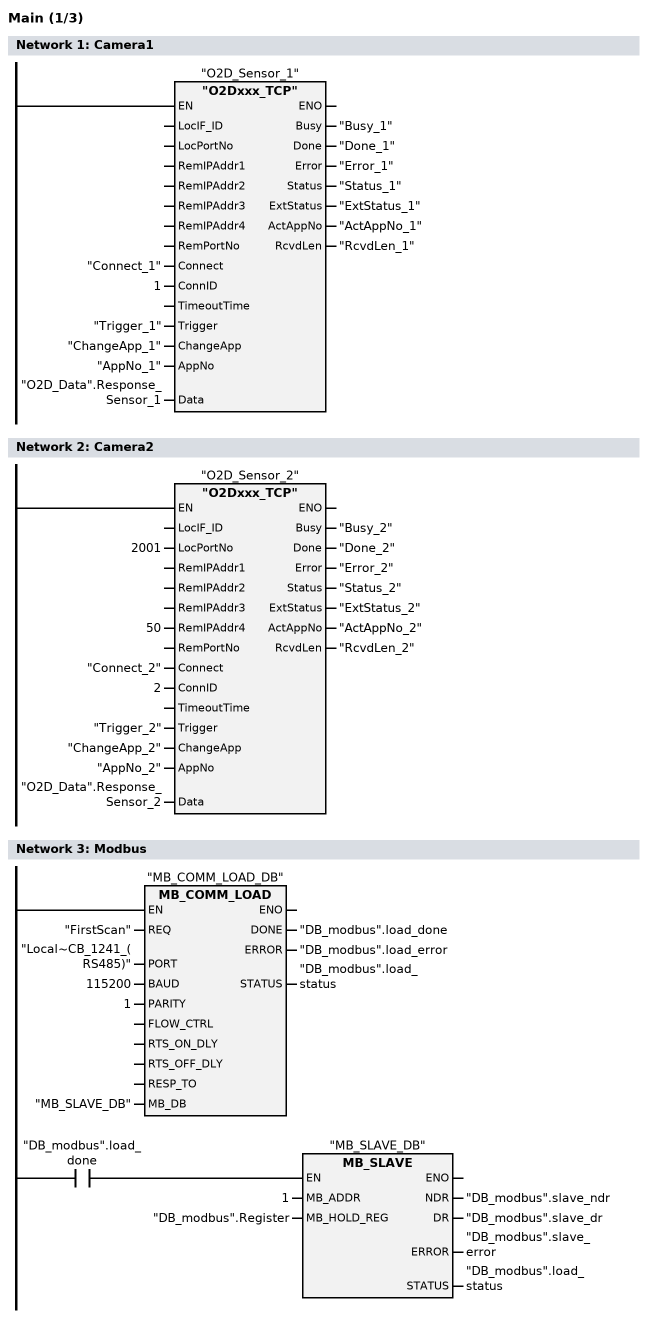
   RUNG wire#powerrail
      "O2D_Sensor_1"(LocIF_ID :=, LocPortNo :=, RemIPAddr1 :=, RemIPAddr2 :=, RemIPAddr3 :=, RemIPAddr4 :=, RemPortNo :=, Connect := "Connect_1", ConnID := 1, TimeoutTime :=, Trigger := "Trigger_1", ChangeApp := "ChangeApp_1", AppNo := "AppNo_1", Data := "O2D_Data".Response_Sensor_1, Busy => "Busy_1", Done => "Done_1", Error => "Error_1", Status => "Status_1", ExtStatus => "ExtStatus_1", ActAppNo => "ActAppNo_1", RcvdLen => "RcvdLen_1")
   END_RUNG
   // the same network as SCL:
   "O2D_Sensor_1"(Connect := "Connect_1",   // "O2Dxxx_TCP"
                  ConnID := 1,
                  Trigger := "Trigger_1",
                  ChangeApp := "ChangeApp_1",
                  AppNo := "AppNo_1",
                  Data := "O2D_Data".Response_Sensor_1,
                  Busy => "Busy_1",
                  Done => "Done_1",
                  Error => "Error_1",
                  Status => "Status_1",
                  ExtStatus => "ExtStatus_1",
                  ActAppNo => "ActAppNo_1",
                  RcvdLen => "RcvdLen_1");
END_REGION

REGION Network 2: Camera2
   RUNG wire#powerrail
      "O2D_Sensor_2"(LocIF_ID :=, LocPortNo := 2001, RemIPAddr1 :=, RemIPAddr2 :=, RemIPAddr3 :=, RemIPAddr4 := 50, RemPortNo :=, Connect := "Connect_2", ConnID := 2, TimeoutTime :=, Trigger := "Trigger_2", ChangeApp := "ChangeApp_2", AppNo := "AppNo_2", Data := "O2D_Data".Response_Sensor_2, Busy => "Busy_2", Done => "Done_2", Error => "Error_2", Status => "Status_2", ExtStatus => "ExtStatus_2", ActAppNo => "ActAppNo_2", RcvdLen => "RcvdLen_2")
   END_RUNG
   // the same network as SCL:
   "O2D_Sensor_2"(LocPortNo := 2001,   // "O2Dxxx_TCP"
                  RemIPAddr4 := 50,
                  Connect := "Connect_2",
                  ConnID := 2,
                  Trigger := "Trigger_2",
                  ChangeApp := "ChangeApp_2",
                  AppNo := "AppNo_2",
                  Data := "O2D_Data".Response_Sensor_2,
                  Busy => "Busy_2",
                  Done => "Done_2",
                  Error => "Error_2",
                  Status => "Status_2",
                  ExtStatus => "ExtStatus_2",
                  ActAppNo => "ActAppNo_2",
                  RcvdLen => "RcvdLen_2");
END_REGION

REGION Network 3: Modbus
   "MB_COMM_LOAD_DB"(REQ := "FirstScan",   // MB_COMM_LOAD
                     PORT := "Local~CB_1241_(RS485)",
                     BAUD := 115200,
                     PARITY := 1,
                     MB_DB := "MB_SLAVE_DB",
                     DONE => "DB_modbus".load_done,
                     ERROR => "DB_modbus".load_error,
                     STATUS => "DB_modbus".load_status);
   IF "DB_modbus".load_done THEN
       "MB_SLAVE_DB"(MB_ADDR := 1,   // MB_SLAVE
                     MB_HOLD_REG := "DB_modbus".Register,
                     NDR => "DB_modbus".slave_ndr,
                     DR => "DB_modbus".slave_dr,
                     ERROR => "DB_modbus".slave_error,
                     STATUS => "DB_modbus".load_status);
   END_IF;
END_REGION

REGION Network 4: Data
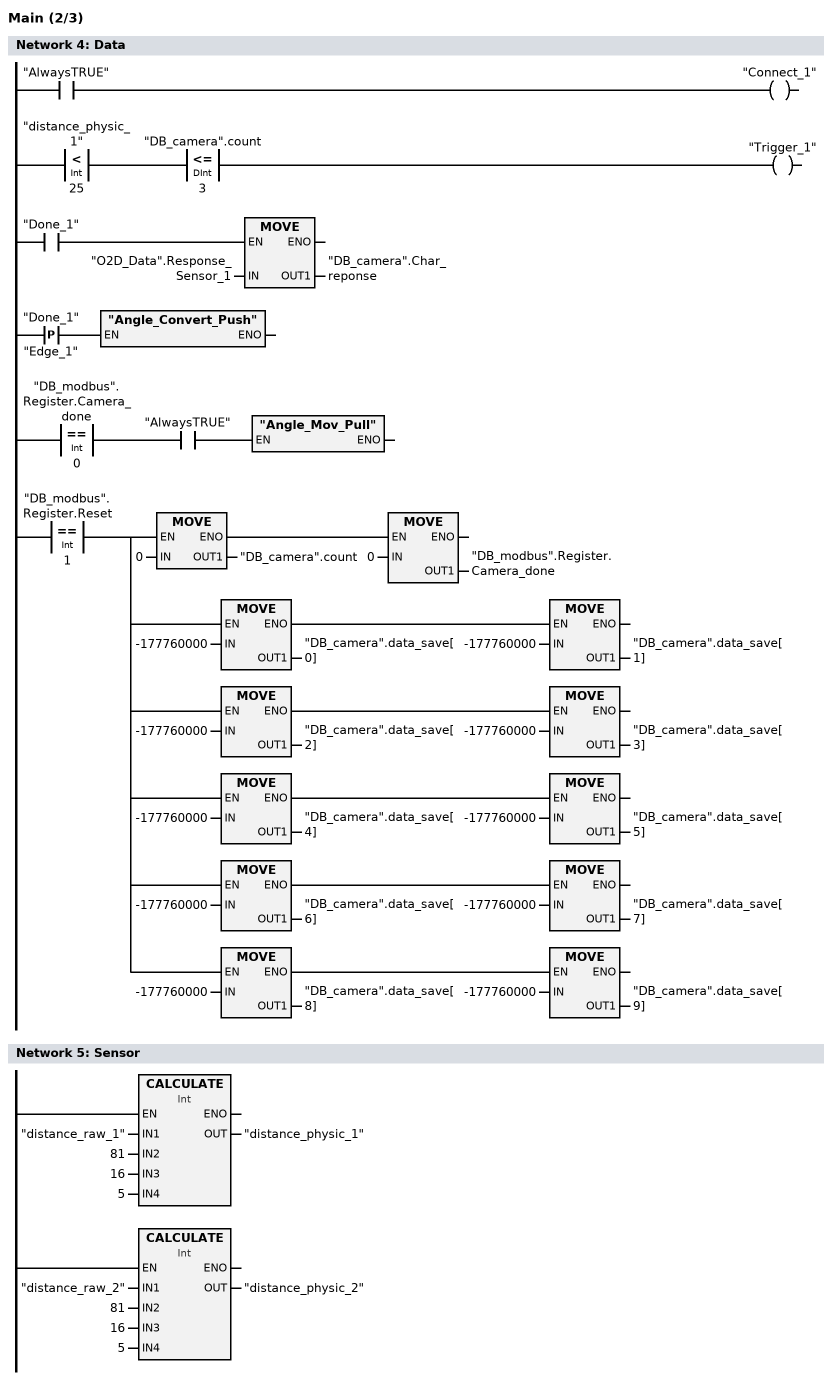
   RUNG wire#powerrail
      Contact( "AlwaysTRUE" )
      Coil( "Connect_1" )
   END_RUNG
   RUNG wire#powerrail
      { S7_Templates := "SrcType := Int" } LT_Contact(in1 := "distance_physic_1", in2 := 25)
      { S7_Templates := "SrcType := DInt" } LE_Contact(in1 := "DB_camera".count, in2 := 3)
      Coil( "Trigger_1" )
   END_RUNG
   RUNG wire#powerrail
      Contact( "Done_1" )
      Move(in := "O2D_Data".Response_Sensor_1, out1 => "DB_camera".Char_reponse)
   END_RUNG
   RUNG wire#powerrail
      P_Contact(operand := "Done_1", bit := "Edge_1")
      "Angle_Convert_Push"()
   END_RUNG
   RUNG wire#powerrail
      { S7_Templates := "SrcType := Int" } EQ_Contact(in1 := "DB_modbus".Register.Camera_done, in2 := 0)
      Contact( "AlwaysTRUE" )
      "Angle_Mov_Pull"()
   END_RUNG
   RUNG wire#powerrail
      { S7_Templates := "SrcType := Int" } EQ_Contact(in1 := "DB_modbus".Register.Reset, in2 := 1)
      wire#w1
      Move(in := 0, out1 => "DB_camera".count)
      Move(in := 0, out1 => "DB_modbus".Register.Camera_done)
   END_RUNG
   RUNG wire#w1
      Move(in := -177760000, out1 => "DB_camera".data_save[0])
      Move(in := -177760000, out1 => "DB_camera".data_save[1])
   END_RUNG
   RUNG wire#w1
      Move(in := -177760000, out1 => "DB_camera".data_save[2])
      Move(in := -177760000, out1 => "DB_camera".data_save[3])
   END_RUNG
   RUNG wire#w1
      Move(in := -177760000, out1 => "DB_camera".data_save[4])
      Move(in := -177760000, out1 => "DB_camera".data_save[5])
   END_RUNG
   RUNG wire#w1
      Move(in := -177760000, out1 => "DB_camera".data_save[6])
      Move(in := -177760000, out1 => "DB_camera".data_save[7])
   END_RUNG
   RUNG wire#w1
      Move(in := -177760000, out1 => "DB_camera".data_save[8])
      Move(in := -177760000, out1 => "DB_camera".data_save[9])
   END_RUNG
   // the same network as SCL:
   "Connect_1" := "AlwaysTRUE";
   "Trigger_1" := ("distance_physic_1" < 25) AND ("DB_camera".count <= 3);
   IF "Done_1" THEN "DB_camera".Char_reponse := "O2D_Data".Response_Sensor_1; END_IF;
   #_w1 := "Done_1" AND NOT "Edge_1";   // rising edge of "Done_1"
   "Edge_1" := "Done_1";
   IF #_w1 THEN "Angle_Convert_Push"(); END_IF;
   IF ("DB_modbus".Register.Camera_done = 0) AND "AlwaysTRUE" THEN "Angle_Mov_Pull"(); END_IF;
   IF "DB_modbus".Register.Reset = 1 THEN
       "DB_camera".count := 0;
       "DB_modbus".Register.Camera_done := 0;
       "DB_camera".data_save[0] := -177760000;
       "DB_camera".data_save[1] := -177760000;
       "DB_camera".data_save[2] := -177760000;
       "DB_camera".data_save[3] := -177760000;
       "DB_camera".data_save[4] := -177760000;
       "DB_camera".data_save[5] := -177760000;
       "DB_camera".data_save[6] := -177760000;
       "DB_camera".data_save[7] := -177760000;
       "DB_camera".data_save[8] := -177760000;
       "DB_camera".data_save[9] := -177760000;
   END_IF;
END_REGION

REGION Network 5: Sensor
   RUNG wire#powerrail
      { S7_Templates := "SrcType := Int"; S7_Expression := "(IN1-IN2)/IN3+IN4" } Calculate(in1 := "distance_raw_1", in2 := 81, in3 := 16, in4 := 5, out => "distance_physic_1")
   END_RUNG
   RUNG wire#powerrail
      { S7_Templates := "SrcType := Int"; S7_Expression := "(IN1-IN2)/IN3+IN4" } Calculate(in1 := "distance_raw_2", in2 := 81, in3 := 16, in4 := 5, out => "distance_physic_2")
   END_RUNG
   // the same network as SCL:
   "distance_physic_1" := ("distance_raw_1"-81)/16+5;
   "distance_physic_2" := ("distance_raw_2"-81)/16+5;
END_REGION

REGION Network 6: Conveyor
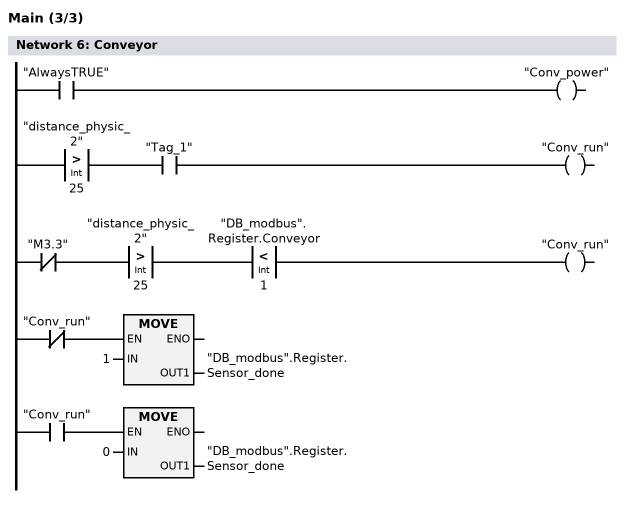
   RUNG wire#powerrail
      Contact( "AlwaysTRUE" )
      Coil( "Conv_power" )
   END_RUNG
   RUNG wire#powerrail
      { S7_Templates := "SrcType := Int" } GT_Contact(in1 := "distance_physic_2", in2 := 25)
      Contact( "Tag_1" )
      Coil( "Conv_run" )
   END_RUNG
   RUNG wire#powerrail
      I_Contact( "M3.3" )
      { S7_Templates := "SrcType := Int" } GT_Contact(in1 := "distance_physic_2", in2 := 25)
      { S7_Templates := "SrcType := Int" } LT_Contact(in1 := "DB_modbus".Register.Conveyor, in2 := 1)
      Coil( "Conv_run" )
   END_RUNG
   RUNG wire#powerrail
      I_Contact( "Conv_run" )
      Move(in := 1, out1 => "DB_modbus".Register.Sensor_done)
   END_RUNG
   RUNG wire#powerrail
      Contact( "Conv_run" )
      Move(in := 0, out1 => "DB_modbus".Register.Sensor_done)
   END_RUNG
   // the same network as SCL:
   "Conv_power" := "AlwaysTRUE";
   "Conv_run" := ("distance_physic_2" > 25) AND "Tag_1";
   "Conv_run" := NOT "M3.3" AND ("distance_physic_2" > 25) AND ("DB_modbus".Register.Conveyor < 1);
   IF NOT "Conv_run" THEN "DB_modbus".Register.Sensor_done := 1; END_IF;
   IF "Conv_run" THEN "DB_modbus".Register.Sensor_done := 0; END_IF;
END_REGION
END_ORGANIZATION_BLOCK